PROGRAM MAIN
VAR
	valve1			: FB_Valve;
	valve2			: FB_Valve;
	valve3			: FB_Valve;
END_VAR

valve1(ib_enable:=TRUE );
valve2(ib_enable:=TRUE );
valve3(ib_enable:=TRUE );

END_PROGRAM

(* stored: Version 1.1.0.1, ProductVersion 3.1.4024.13
   POU MAIN: Id {73efd3e7-4f6b-44ac-9afb-94da7e292ce7}, SpecialFunc None *)
